Universal Robots PolyScope program: modbustest-archive.urp

Program modbustest-archive (installation=default directory=/programs createdIn=5.11.5.1010327 lastSavedIn=5.11.5.1010327 robotSerialNumber=20215500677)
Calibrated DH parameters: a=[0.000204, -0.239222, -0.391845, -0.000001, 0.000022, 0]; d=[0.162722, -355.808559, 353.37206, 2.570385, 0.099741, 0.099629]; alpha=[1.571124, 0.000988, 0.008295, 1.568963, -1.570303, 0]; deltaTheta=[0, -0.973091, 7.204745, 0.05153, 0, 0]
BeforeStart
  Set ExpressionOutput pin=ROBOT_SENDING; expression=False
  Script file /programs/cube/set_conveyor_params.script
    | def Set_Conveyor_Params(velocity, acceleration):
    | modbus_set_output_signal("ROBOT_SENDING", True, False)
    | modbus_set_output_register("VELOCITY", velocity, False)
    | modbus_set_output_register("ACCELERATION", acceleration, False)
    | sleep(.05)
    | modbus_set_output_signal("ROBOT_SENDING", False, False)
    | end
  Script file /programs/cube/set_motion_mode.script
    | def Set_Motion_Mode(modeString):
    |   if modeString == "distance":
    |     modbus_set_output_register("MOTION_MODE", 0, False)
    |   elif modeString == "position":
    |     modbus_set_output_register("MOTION_MODE", 1, False)
    |   elif modeString == "continuous":
    |     modbus_set_output_register("MOTION_MODE", 2, False)
    |   elif modeString == "idle":
    |     modbus_set_output_register("MOTION_MODE", 3, False)
    |   else:
    |     modbus_set_output_register("MOTION_MODE", 3, False)
    |   end
    | 
    | end
  Script file /programs/cube/position_move.script
    | def Move_Position(position):
    |   modbus_set_output_signal("ROBOT_SENDING", True, False)
    |   Set_Motion_Mode("position")
    |   modbus_set_output_register("POSITION", position, False)
    |   Set_Request_Id()
    |   sleep(.05)
    |   modbus_set_output_signal("ROBOT_SENDING", False, False)
    | end
  Script file /programs/cube/distance_move.script
    | def Move_Distance(distance):
    |   modbus_set_output_signal("ROBOT_SENDING", True, False)
    |   Set_Motion_Mode("distance")
    |   distance = Inches_To_Steps(distance)
    |   if distance < 0:
    |   distance = distance * -1
    |   modbus_set_output_signal("DIRECTION", False, False)
    |   else:
    |   modbus_set_output_signal("DIRECTION", True, False)
    |   end
    |   modbus_set_output_register("DISTANCE", distance, False)
    |   Set_Request_Id()
    |   sleep(.05)
    |   modbus_set_output_signal("ROBOT_SENDING", False, False)
    |   mode = modbus_get_signal_status("MOTION_MODE", False)
    |   while (mode  != 3):
    |     mode = modbus_get_signal_status("MOTION_MODE", False)
    |     sync()
    |   end
    | end
  Script file /programs/cube/mm_move.script
    | def Conveyor_Move_mm(distance):
    |   modbus_set_output_signal("ROBOT_SENDING", True, False)
    |   modbus_set_output_register("MOTION_MODE", 0, False)
    |   distance = mm_to_steps(distance)
    |   if distance < 0:
    |   distance = distance * -1
    |   modbus_set_output_signal("DIRECTION", False, False)
    |   else:
    |   modbus_set_output_signal("DIRECTION", True, False)
    |   end
    |   modbus_set_output_register("DISTANCE", distance, False)
    |   Set_Request_Id()
    |   modbus_set_output_signal("ROBOT_SENDING", False, False)
    | end
  Script file /programs/cube/continuous_move.script
    | def Move_Continuous(direction):
    |   modbus_set_output_signal("ROBOT_SENDING", True, False)
    |   Set_Motion_Mode("continuous")
    |   if direction == "forward":
    |   modbus_set_output_signal("DIRECTION", True, False)
    |   else:
    |   modbus_set_output_signal("DIRECTION", False, False)
    |   end
    |   Set_Request_Id()
    |   sleep(.05)
    |   modbus_set_output_signal("ROBOT_SENDING", False, False)
    | end
  Script file /programs/cube/idle_move.script
    | def Move_Idle():
    |   modbus_set_output_signal("ROBOT_SENDING", True, False)
    |   Set_Motion_Mode("idle")
    |   Set_Request_Id()
    |   sleep(.05)
    |   modbus_set_output_signal("ROBOT_SENDING", False, False)
    | end
  Script file /programs/cube/request_id.script
    | def Set_Request_Id():
    | id = floor(random()*65000)
    | modbus_set_output_register("REQUEST_ID", id, False)
    | end
  Script file /programs/cube/steps_per_inch.script
    | def Inches_To_Steps(distance):
    | mm = distance*25.4
    | return mm_to_steps(mm)
    | end
  Script file /programs/cube/mm_to_steps.script
    | def mm_to_steps(distance):
    | teeth = 28
    | pitch = 2
    | degreesPerStep = 1.8
    | microsteps = 8
    | adjustment = 400/381
    | microStepsPerMm = 360 / teeth  / degreesPerStep / pitch * microsteps * adjustment
    | return floor(distance * microStepsPerMm)
    | end
  Script: Set_Conveyor_Params(1600, 16000)
  Script: Move_Idle()
  Script file /programs/select_job.script
    | def read_job():
    | job = modbus_get_signal_status("JOB", False)
    | #1 - cube, 2 - browser,  3 - 45
    | #4 - stereocab 2, 5 - sc 3, 6 - sc4
    | if job == 1:
    |   width = 362
    |   height = 362
    |   depth = 349
    | elif job == 2:
    |   width = 362
    |   height = 362
    |   depth = 235
    | elif job == 3:
    |   width = 724
    |   height = 235
    |   depth = 349
    | elif job == 4:
    |   width = 724
    |   height = 235
    |   depth = 349
    | elif job == 5:
    |   width = 1086
    |   height = 235
    |   depth = 349
    | elif job == 6:
    |   width = 1448
    |   height = 235
    |   depth = 349
    | end
    | sleep(.2)
    | end
  loaded := 0
  dried := False
  Set ExpressionOutput pin=BRUSH_ON; expression=False
  SuppressedNode
    MoveJ speed 60 deg/s, acceleration 80 deg/s^2 (useActiveTCP=false) tcp=SandTCP; feature=Base
      Waypoint Sand_Base: TCP in base x=-331.002 y=208.013 z=654.466 mm, rx=0.0315 ry=-0.0315 rz=-1.5705 rad; joints [-61.396, -81.213, 112.495, 86.07, -50.257, -128.662] deg; TCP offset x=1.003 y=125.541 z=104.154 mm, rx=-0.7854 ry=0 rz=0 rad
Robot Program (runOnlyOnce=false)
  MoveJ speed 60 deg/s, acceleration 80 deg/s^2 (useActiveTCP=false) tcp=SandTCP; feature=Base
    Waypoint Sand_Base: TCP in base x=-331.002 y=208.013 z=654.466 mm, rx=0.0315 ry=-0.0315 rz=-1.5705 rad; joints [-61.396, -81.213, 112.495, 86.07, -50.257, -128.662] deg
  SuppressedNode
    Loop While (checkContinuously=true) expression=RUN==False
      If MOTION_MODE ≠ 3
        Script: Move_Idle()
      If FEED_CONVEYOR≟ True (checkContinuously=true)
        Set ExpressionOutput pin=FEED_CONVEYOR; expression=False
      Script: sync()
  SuppressedNode
    Folder Load Workpiece [hidden by the author, left out]
  SuppressedNode
    If RUN == True
      Script: read_job()
      Folder Sand [hidden by the author, left out]
      Folder 45 Sand [hidden by the author, left out]
      Folder SC 3 and 4 Sand
        If JOB == 5 or JOB == 6
          Script: Conveyor_Move_mm((width-12)/2)
          Wait Condition expression=SERVER_STATE==1
          MoveL speed 50 mm/s, acceleration 500 mm/s^2 (useActiveTCP=false) tcp=SandTCP; feature=Base
            MoveDirectionNode (selectedDirection=XMinus)
              Until DISTANCE (allowActions=false deceleration=3 distanceNodeType=STOP) Distance=0.085; motionParameters(blendRadius=0)
            MoveDirectionNode (selectedDirection=ZPlus toolParams=0.05, 0.5)
              Until TOOL_CONTACT_DETECTION (allowActions=false retraction=0 decelerationAcceleration=3 decelerationAngularAcceleration=34.906585)
            URCap Finishing Tool Control (Robotiq_Copilot, Robotiq Inc.) dataModel(ToolOutputNameKey=SanderOn, HackTriggeringContributionIsDefinedMethodKey=true)
            Force Simple feature=Base; selection=[0, 0, 1, 0, 0, 0]; wrench=[0, 0, 10, 0, 0, 0]; limitsForce=[0.15, 0.15, 0.15, 1.047198, 1.047198, 1.047198]; limitsMotion=[0.1, 0.1, 0.1, 0.349066, 0.349066, 0.349066]
              MoveDirectionNode (selectedDirection=XMinus)
                Until DISTANCE (allowActions=false deceleration=3 distanceNodeType=STOP) Distance=0.08; motionParameters(blendRadius=0)
              URCap Finishing Tool Control (Robotiq_Copilot, Robotiq Inc.) dataModel(FinishingToolStateKey=false, ToolOutputNameKey=SanderOn, HackTriggeringContributionIsDefinedMethodKey=true)
            MoveDirectionNode (selectedDirection=ZMinus)
              Until DISTANCE (allowActions=false deceleration=3 distanceNodeType=STOP) Distance=0.05; motionParameters(blendRadius=0)
            Script: Conveyor_Move_mm(-(width-12)/2)
            Wait Condition expression=SERVER_STATE==1
      Folder Spray Vertical [hidden by the author, left out]
      Folder 45 Spray [hidden by the author, left out]
      Folder SC 3 and 4 Spray [hidden by the author, left out]
      Folder Cube [hidden by the author, left out]
      MoveJ speed 60 deg/s, acceleration 80 deg/s^2 (useActiveTCP=false) tcp=SandTCP; feature=Base
        Waypoint Sand_Base: TCP in base x=-331.002 y=208.013 z=654.466 mm, rx=0.0315 ry=-0.0315 rz=-1.5705 rad; joints [-61.396, -81.213, 112.495, 86.07, -50.257, -128.662] deg
      Folder Clean Spray
        MoveJ speed 60 deg/s, acceleration 80 deg/s^2 (useActiveTCP=false) tcp=SandTCP; feature=Base
          Waypoint Sand_Base: TCP in base x=-331.002 y=208.013 z=654.466 mm, rx=0.0315 ry=-0.0315 rz=-1.5705 rad; joints [-61.396, -81.213, 112.495, 86.07, -50.257, -128.662] deg
          Waypoint Clean_Brush: TCP in base x=-466.566 y=462.734 z=411.72 mm, rx=-1.4127 ry=-0.6163 rz=0.894 rad; joints [-66.849, -61.854, 103.876, 85.813, -75.713, -328.962] deg
          Set ExpressionOutput pin=BRUSH_ON; expression=True
          MoveL speed 50 mm/s, acceleration 500 mm/s^2 (useActiveTCP=true) feature=Base
            MoveDirectionNode (selectedDirection=ZPlus)
              Until DISTANCE (allowActions=false deceleration=3 distanceNodeType=STOP) Distance=0.008; motionParameters(blendRadius=0)
          Timer (action=Start) variable(name=timer_brush)
      If dried≟ False
        Folder Dry [hidden by the author, left out]
      Else 
        Folder Unload Workpiece [hidden by the author, left out]
  Folder Motion Test
    Script: Conveyor_Move_mm(width)
    Wait Condition expression=SERVER_STATE == 1
    SuppressedNode
      Wait Sleep waitTime=2
  Script: sync()
Thread Thread_1 (runOnlyOnce=false)
  If RUN == False (checkContinuously=true)
    If MOTION_MODE ≠3 (checkContinuously=true)
      Script: Move_Idle()
    If FEED_CONVEYOR≟ True (checkContinuously=true)
      Set ExpressionOutput pin=FEED_CONVEYOR; expression=False
    Script: sync()
  Else 
    Script: sync()
Thread Thread_2 (runOnlyOnce=false)
  If timer_brush > 30 (checkContinuously=true)
    Set ExpressionOutput pin=BRUSH_ON; expression=False
    Timer (action=Stop) variable=timer_brush
    Timer (action=Reset) variable=timer_brush
  Script: sync()
